{attribute 'Tc2GvlVarNames'}
VAR_GLOBAL
	Shark: BOOL;

(* MFSC *)

	Source_MaxPhotonics										:Data_Laser; 

	PLC_Prog_Power_Watt_Max										: UDINT := 6000; 		(* Watt *) (* 0... 6000*)	(* OK *)
	PLC_Prog_Power_Watt_Target									: UDINT := 0; 			(* Watt *) (* 0... 6000*)	(* OK *)
	(***********************************************************************************************************************)
	PLC_Prog_Per_Cent_Of_Duty_Cycle_Max							: UDINT := 100;		(* 0...100% *)			(* OK *)
	PLC_Prog_Per_Cent_Of_Duty_Cycle_Target						: UDINT := 0;			(* 0...100% *)			(* OK *)
	(***********************************************************************************************************************)
	PLC_Prog_Frequency_0_20000Hz_Max							: UDINT := 20000;		(* Hz *) (* 0... 20 000 *)	(* OK *)
	PLC_Prog_Frequency_0_20000Hz_Target							: UDINT := 0; 			(* Hz *) (* 0... 20 000Hz *)(* OK *)
	(***********************************************************************************************************************)

	Prog_Cutting_Mode										: BOOL := TRUE;
	Prog_Marking_Mode										: BOOL := FALSE;                                                  	
	Prog_Secu_Source_OK										: BOOL;						(* OK *)                                              	
	Prog_Annul_Defaut_Source								: BOOL;						(* OK *)
	Prog_Source_Prete_Pour_Decoupe							: BOOL;                                                          
	Prog_Defaut_power_Watt_Target							: BOOL;						(* OK *)
	Prog_Defaut_Perc_Cent_Of_Laser_Output_Power_FeedBack	: BOOL;						(* OK *)
	Prog_Defaut_Per_Cent_Of_Duty_Cycle_Target				: BOOL;						(* OK *)
	Prog_Defaut_Laser_Frequency_Of_PWM_Wave_Target			: BOOL;						(* OK *)
	Prog_Defaut_Status_2									: BOOL;						(* OK *)
	Prog_Defaut_Status_3									: BOOL;						(* OK *)
	Prog_Defaut_Status_4									: BOOL;						(* OK *)                                                   	
	Prog_Defaut_Source_Laser								: BOOL;						(* OK *)
	
	OUT_Perc_Duty_PWM	AT%Q*:UINT;
	OUT_Freq_PWM		AT%Q*:UDINT;
	
END_VAR

(* stored: Version 1.1.0.1
   GVL IO_SOURCE_MAXPHOTONICS: Id {e72f5ffe-2adf-4f12-b359-592dff2a5a24} *)
